(* Logix 5000 project; controller Sucrose_Main Emulate 5570 rev 20.12; software revision 20.01; part 30 of 30 *)
(* tags used below, declared in another part *)
   Alarm_ACK_Master_Timer : TIMER;
   DI_E23_3 : ALIAS FOR FLX_E23:3:I;   // Discrete Input EN2T_FLX 192.168.1.23
   DO_E24_5 : ALIAS FOR FLX_E24:5:O;   // Discrete Output EN2T_FLX 192.168.1.24
   DO_E24_6 : ALIAS FOR FLX_E24:6:O;   // Discrete Output EN2T_FLX 192.168.1.24
   HTR760201_AOI : QSI_Discrete_Device;   // HTR-76-02-01 SUCROSE TANK #2 UTILITY HOT WATER ELECTRIC HEATER ENABLE
   HTR760301_AOI : QSI_Discrete_Device;   // HTR-76-03-01 SUCROSE TANK #3 UTILITY HOT WATER ELECTRIC HEATER ENABLE
   Sucrose_MM_Enable : BOOL;
   SucroseTanks : Area_Program;
   SV931101_AOI : QSI_Discrete_Device;   // SV-93-11-01 STERILE AIR AUTO VENT FOR FLT-93-11-01 SOLENOID VALVE
   SV931102_AOI : QSI_Discrete_Device;   // SV-93-11-02 STERILE AIR AUTO DRAIN FOR FLT-93-11-01 SOLENOID VALVE
   SV931201_AOI : QSI_Discrete_Device;   // SV-93-12-01 STERILE AIR AUTO VENT FOR FLT-93-12-01 SOLENOID VALVE
   SV931202_AOI : QSI_Discrete_Device;   // SV-93-12-02 STERILE AIR AUTO DRAIN FOR FLT-93-12-02 SOLENOID VALVE
   SV931301_AOI : QSI_Discrete_Device;   // SV-93-13-01 STERILE AIR AUTO VENT FOR FLT-93-13-01 SOLENOID VALVE
   SV931302_AOI : QSI_Discrete_Device;   // SV-93-13-02 STERILE AIR AUTO DRAIN FOR FLT-93-13-02 SOLENOID VALVE
(* TanksArea_EN2T_IO_Discrete_DO_E24_5, continued *)

ROUTINE _01_HTR760201   (* ladder *)
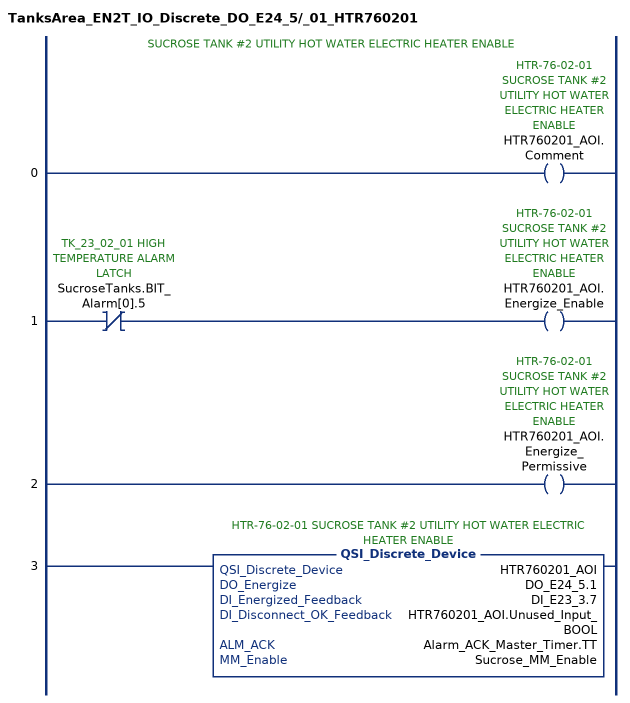
   // SUCROSE TANK #2 UTILITY HOT WATER ELECTRIC HEATER ENABLE
   0: OTE(HTR760201_AOI.Comment);
   1: XIO(SucroseTanks.BIT_Alarm[0].5)OTE(HTR760201_AOI.Energize_Enable);
   2: OTE(HTR760201_AOI.Energize_Permissive);
   3: QSI_Discrete_Device(HTR760201_AOI,DO_E24_5.1,DI_E23_3.7,HTR760201_AOI.Unused_Input_BOOL,Alarm_ACK_Master_Timer.TT,Sucrose_MM_Enable);
END_ROUTINE

ROUTINE _02_HTR760301   (* ladder *)
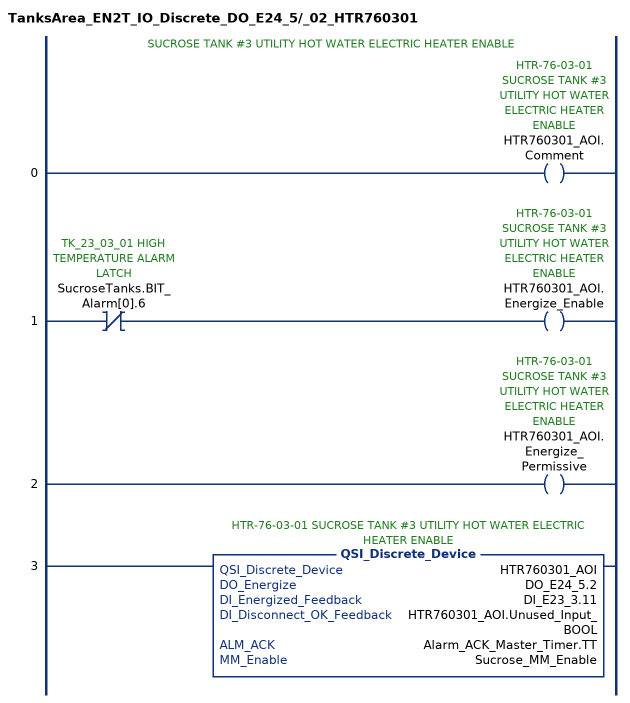
   // SUCROSE TANK #3 UTILITY HOT WATER ELECTRIC HEATER ENABLE
   0: OTE(HTR760301_AOI.Comment);
   1: XIO(SucroseTanks.BIT_Alarm[0].6)OTE(HTR760301_AOI.Energize_Enable);
   2: OTE(HTR760301_AOI.Energize_Permissive);
   3: QSI_Discrete_Device(HTR760301_AOI,DO_E24_5.2,DI_E23_3.11,HTR760301_AOI.Unused_Input_BOOL,Alarm_ACK_Master_Timer.TT,Sucrose_MM_Enable);
END_ROUTINE

ROUTINE MainRoutine   (* ladder *)
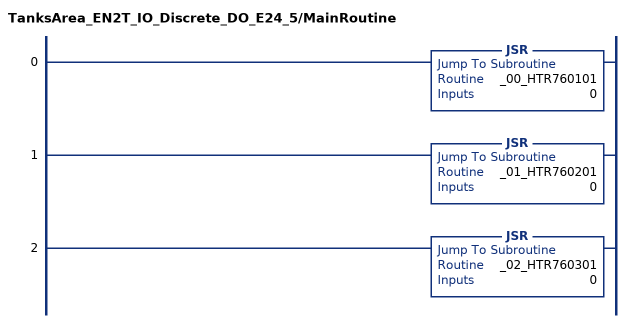
   0: JSR(_00_HTR760101,0);
   1: JSR(_01_HTR760201,0);
   2: JSR(_02_HTR760301,0);
END_ROUTINE
END_PROGRAM

PROGRAM TanksArea_EN2T_IO_Discrete_DO_E24_6   (* main routine MainRoutine *)

ROUTINE _00_SV931101   (* ladder *)
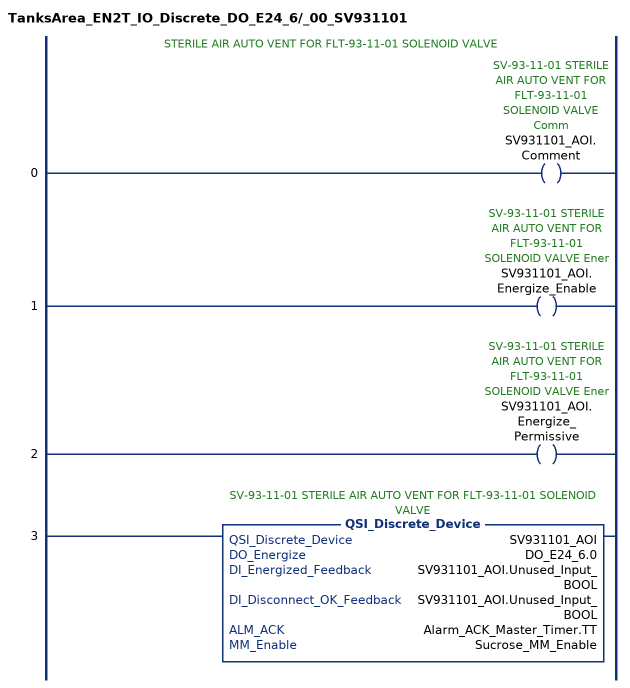
   // STERILE AIR AUTO VENT FOR FLT-93-11-01 SOLENOID VALVE
   0: OTE(SV931101_AOI.Comment);
   1: OTE(SV931101_AOI.Energize_Enable);
   2: OTE(SV931101_AOI.Energize_Permissive);
   3: QSI_Discrete_Device(SV931101_AOI,DO_E24_6.0,SV931101_AOI.Unused_Input_BOOL,SV931101_AOI.Unused_Input_BOOL,Alarm_ACK_Master_Timer.TT,Sucrose_MM_Enable);
END_ROUTINE

ROUTINE _01_SV931102   (* ladder *)
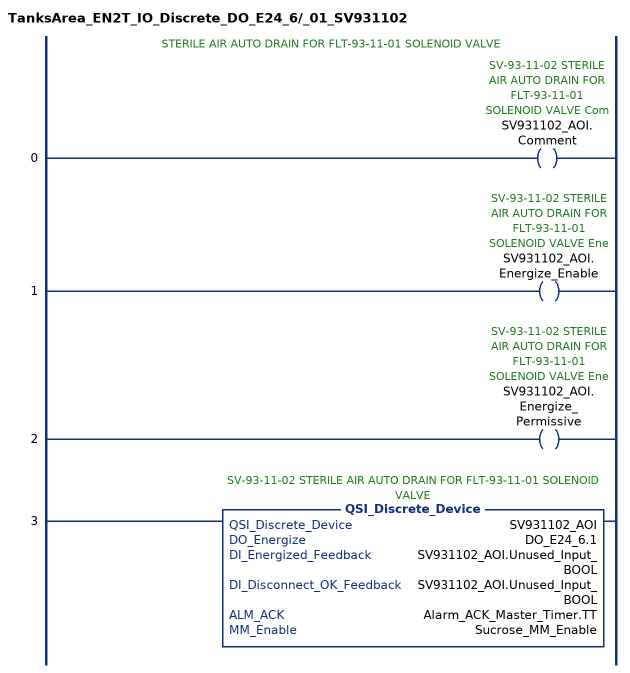
   // STERILE AIR AUTO DRAIN FOR FLT-93-11-01 SOLENOID VALVE
   0: OTE(SV931102_AOI.Comment);
   1: OTE(SV931102_AOI.Energize_Enable);
   2: OTE(SV931102_AOI.Energize_Permissive);
   3: QSI_Discrete_Device(SV931102_AOI,DO_E24_6.1,SV931102_AOI.Unused_Input_BOOL,SV931102_AOI.Unused_Input_BOOL,Alarm_ACK_Master_Timer.TT,Sucrose_MM_Enable);
END_ROUTINE

ROUTINE _02_SV931201   (* ladder *)
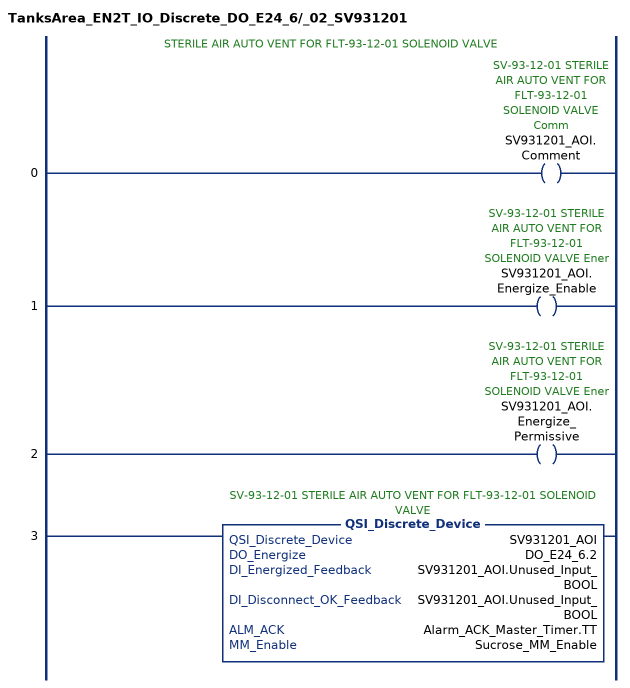
   // STERILE AIR AUTO VENT FOR FLT-93-12-01 SOLENOID VALVE
   0: OTE(SV931201_AOI.Comment);
   1: OTE(SV931201_AOI.Energize_Enable);
   2: OTE(SV931201_AOI.Energize_Permissive);
   3: QSI_Discrete_Device(SV931201_AOI,DO_E24_6.2,SV931201_AOI.Unused_Input_BOOL,SV931201_AOI.Unused_Input_BOOL,Alarm_ACK_Master_Timer.TT,Sucrose_MM_Enable);
END_ROUTINE

ROUTINE _03_SV931202   (* ladder *)
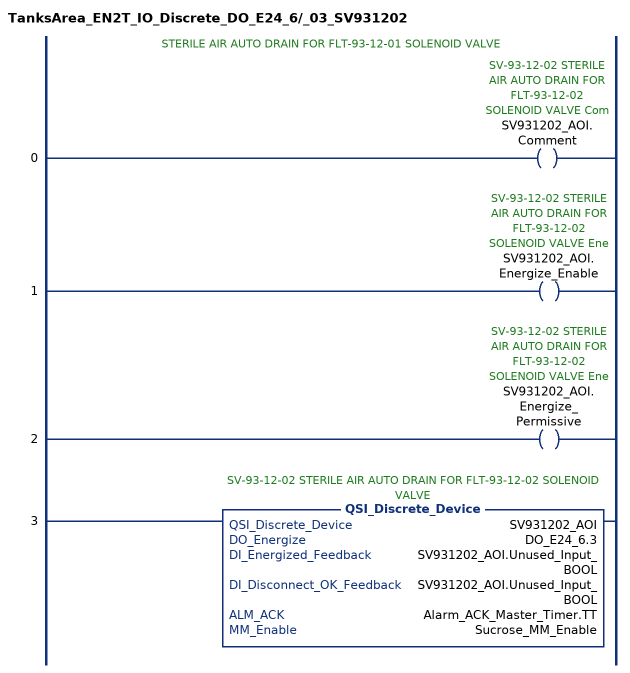
   // STERILE AIR AUTO DRAIN FOR FLT-93-12-01 SOLENOID VALVE
   0: OTE(SV931202_AOI.Comment);
   1: OTE(SV931202_AOI.Energize_Enable);
   2: OTE(SV931202_AOI.Energize_Permissive);
   3: QSI_Discrete_Device(SV931202_AOI,DO_E24_6.3,SV931202_AOI.Unused_Input_BOOL,SV931202_AOI.Unused_Input_BOOL,Alarm_ACK_Master_Timer.TT,Sucrose_MM_Enable);
END_ROUTINE

ROUTINE _04_SV931301   (* ladder *)
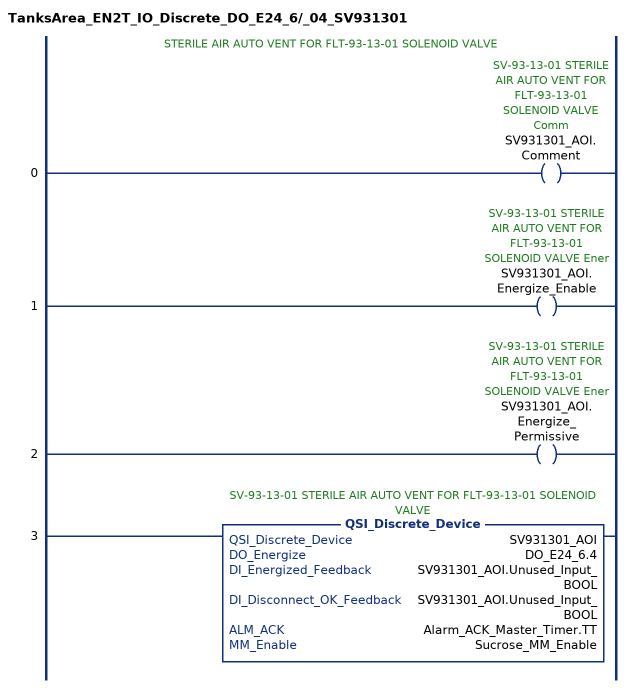
   // STERILE AIR AUTO VENT FOR FLT-93-13-01 SOLENOID VALVE
   0: OTE(SV931301_AOI.Comment);
   1: OTE(SV931301_AOI.Energize_Enable);
   2: OTE(SV931301_AOI.Energize_Permissive);
   3: QSI_Discrete_Device(SV931301_AOI,DO_E24_6.4,SV931301_AOI.Unused_Input_BOOL,SV931301_AOI.Unused_Input_BOOL,Alarm_ACK_Master_Timer.TT,Sucrose_MM_Enable);
END_ROUTINE

ROUTINE _05_SV931302   (* ladder *)
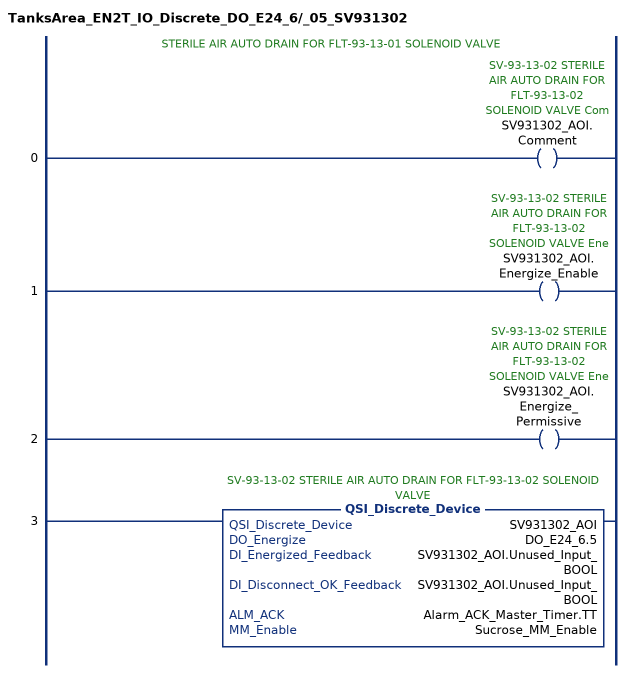
   // STERILE AIR AUTO DRAIN FOR FLT-93-13-01 SOLENOID VALVE
   0: OTE(SV931302_AOI.Comment);
   1: OTE(SV931302_AOI.Energize_Enable);
   2: OTE(SV931302_AOI.Energize_Permissive);
   3: QSI_Discrete_Device(SV931302_AOI,DO_E24_6.5,SV931302_AOI.Unused_Input_BOOL,SV931302_AOI.Unused_Input_BOOL,Alarm_ACK_Master_Timer.TT,Sucrose_MM_Enable);
END_ROUTINE

ROUTINE MainRoutine   (* ladder *)
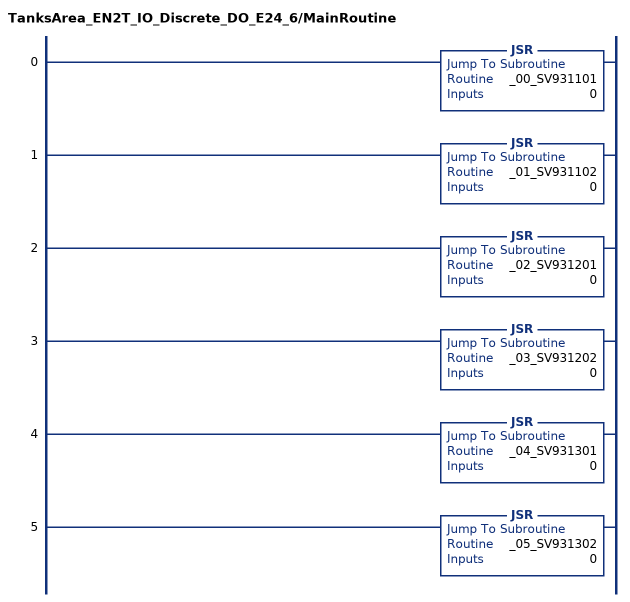
   0: JSR(_00_SV931101,0);
   1: JSR(_01_SV931102,0);
   2: JSR(_02_SV931201,0);
   3: JSR(_03_SV931202,0);
   4: JSR(_04_SV931301,0);
   5: JSR(_05_SV931302,0);
END_ROUTINE
END_PROGRAM
